{attribute 'linkalways'} 
{attribute 'no_explicit_call' := 'This FB is a CLASS and must be accessed using methods or properties'}
{attribute 'enable_dynamic_creation'}
FUNCTION_BLOCK PUBLIC ListNode EXTENDS Disposable IMPLEMENTS I_ListNode
VAR
	pBuffer : POINTER TO BYTE;
	bufferSize : UDINT;
END_VAR

METHOD PRIVATE CopyBufferToDestination
VAR_INPUT
	DestinationAddress : PVOID;
END_VAR
MEMCPY(DestinationAddress, pBuffer, bufferSize);
END_METHOD

METHOD PRIVATE CopySourceToBuffer
VAR_INPUT
	SourceAddress : PVOID;
END_VAR
MEMCPY(pBuffer, SourceAddress, bufferSize);
END_METHOD

METHOD PRIVATE CreateBuffer
VAR_INPUT
	SizeInBytes : UDINT;
END_VAR
bufferSize := SizeInBytes;
pBuffer := __NEW(BYTE, SizeInBytes);
END_METHOD

PROPERTY PUBLIC DataSize : UDINT
GET
DataSize := bufferSize;
END_GET
END_PROPERTY

METHOD PRIVATE DestroyBuffer
VAR_INPUT
END_VAR
IF pBuffer = 0 THEN
	RETURN;
END_IF

__DELETE(pBuffer);
bufferSize := 0;
END_METHOD

METHOD PUBLIC Equals : BOOL
VAR_INPUT
	Symbol : ANY;
END_VAR
IF pBuffer = 0 THEN
	RETURN;
END_IF

IF bufferSize <> DINT_TO_UDINT(Symbol.diSize) THEN
	RETURN;
END_IF

Equals := memcmp(Symbol.pValue, pBuffer, bufferSize) = 0;
END_METHOD

METHOD FB_exit : BOOL
VAR_INPUT
	bInCopyCode : BOOL; // if TRUE, the exit method is called for exiting an instance that is copied afterwards (online change).
END_VAR
IF bInCopyCode THEN
	RETURN;
END_IF

DestroyBuffer();
END_METHOD

METHOD FB_init : BOOL
VAR_INPUT
	bInitRetains : BOOL; // if TRUE, the retain variables are initialized (warm start / cold start)
	bInCopyCode : BOOL;  // if TRUE, the instance afterwards gets moved into the copy code (online change)
	Source : ANY;
END_VAR
CreateBuffer(DINT_TO_UDINT(Source.diSize));
CopySourceToBuffer(Source.pValue);
END_METHOD

METHOD TryGet : BOOL
VAR_INPUT
	Destination	: ANY;
END_VAR
TryGet := TryGetTo(Destination.pValue, DINT_TO_UDINT(Destination.diSize));
END_METHOD

METHOD TryGetTo : BOOL
VAR_INPUT
	DestinationAddress : PVOID;
	DestinationSize : UDINT;
END_VAR
IF pBuffer = 0 THEN
	RETURN;
END_IF

IF bufferSize <> DestinationSize THEN
	RETURN;
END_IF

CopyBufferToDestination(DestinationAddress);
TryGetTo := TRUE;
END_METHOD

END_FUNCTION_BLOCK

(* stored: Version 1.1.0.1, ProductVersion 3.1.4024.12
   POU ListNode: Id {93aff3e5-d86d-0eb6-0d8e-016cd0fdea02}, SpecialFunc None
   Folder Constructor: Id {1526a92e-19f1-0fe1-09d7-80d02393ef8d}
   Folder Destructor: Id {8635e0ca-71df-09d6-2ada-cee05bc00bc5}
   Folder Private: Id {3addb6b1-98c9-07b3-34b0-345460af3fa0}
   Method CopyBufferToDestination: Id {aaf00d0e-1e7b-026b-0d7f-50f5d372c577}
   Method CopySourceToBuffer: Id {9f681f1c-3ad2-0c44-1605-08c8b1585ce3}
   Method CreateBuffer: Id {781440e5-6ab8-04a3-3511-cb7474572f88}
   Property DataSize: Id {c5ed3b8f-bc1e-0103-271c-cc1431f210db}
   Get Get: Id {c005743d-a85e-0126-0134-a309f0a75ec6}
   Method DestroyBuffer: Id {d99d397b-4d70-01c7-0296-c4ab28a2f74e}
   Method Equals: Id {9bedbc6e-acf9-0a32-2ec4-f48090c273a7}
   Method FB_exit: Id {c53c1ac2-3017-0b39-0847-5e9d150a844f}
   Method FB_init: Id {c8894410-f0ce-05e1-1ee2-98fd8e57c229}
   Method TryGet: Id {de5e3775-17a7-0c52-2901-d863a9097e33}
   Method TryGetTo: Id {664725f6-d390-0ae4-37fe-7203f4e7025e} *)
